TYPE ST_Wedge :
STRUCT
    fLength : LREAL; // [mm]
    fThicknessRange : ARRAY[1..2] OF LREAL; // [mm]
END_STRUCT
END_TYPE

(* stored: Version 1.1.0.1
   DUT ST_Wedge: Id {035ff6df-d87c-42df-97e7-ae575085b871} *)
